// Mitsubishi GX Works2 project: BookEX6_35 Struct   PLC: Q13UDV

// global labels: Global
VAR_GLOBAL
  bVar0 AT M5000 : BOOL;
  abArray0 AT M5010 : ARRAY [0..49] OF BOOL;
  sStr0 AT D5000 : STRING[199];
  sStr1 AT D5100 : STRING[199];
  sStr2 AT D5200 : STRING[199];
  sStr3 AT D5300 : STRING[199];
  sStr4 AT D5400 : STRING[199];
  sStr5 AT D5500 : STRING[199];
  sStr6 AT D5600 : STRING[199];
  sStr7 AT D5700 : STRING[199];
  sStr8 AT D5800 : STRING[199];
  sStr9 AT D5900 : STRING[199];
  iVar0 AT D4500 : INT;
  iVar1 AT D4501 : INT;
  iVar2 AT D4502 : INT;
  iVar3 AT D4503 : INT;
  iVar4 AT D4504 : INT;
  iVar5 AT D4505 : INT;
  iVar6 AT D4506 : INT;
  iVar7 AT D4507 : INT;
  iVar8 AT D4508 : INT;
  iVar9 AT D4509 : INT;
  dVar0 AT D4510 : DINT;
  dVar1 AT D4512 : DINT;
  dVar2 AT D4514 : DINT;
  dVar3 AT D4516 : DINT;
  dVar4 AT D4518 : DINT;
  dVar5 AT D4520 : DINT;
  dVar6 AT D4522 : DINT;
  dVar7 AT D4524 : DINT;
  dVar8 AT D4526 : DINT;
  dVar9 AT D4528 : DINT;
  wVar0 AT D4530 : WORD;
  wVar1 AT D4531 : WORD;
  wVar2 AT D4532 : WORD;
  wVar3 AT D4533 : WORD;
  wVar4 AT D4534 : WORD;
  wVar5 AT D4535 : WORD;
  wVar6 AT D4536 : WORD;
  wVar7 AT D4537 : WORD;
  wVar8 AT D4538 : WORD;
  wVar9 AT D4539 : WORD;
  dwVar0 AT D4540 : DWORD;
  dwVar1 AT D4542 : DWORD;
  dwVar2 AT D4544 : DWORD;
  dwVar3 AT D4546 : DWORD;
  dwVar4 AT D4548 : DWORD;
  dwVar5 AT D4550 : DWORD;
  dwVar6 AT D4552 : DWORD;
  dwVar7 AT D4554 : DWORD;
  dwVar8 AT D4556 : DWORD;
  dwVar9 AT D4558 : DWORD;
  fsVar0 AT D4560 : REAL;
  fsVar1 AT D4562 : REAL;
  fsVar2 AT D4564 : REAL;
  fsVar3 AT D4566 : REAL;
  fsVar4 AT D4568 : REAL;
  fsVar5 AT D4570 : REAL;
  fsVar6 AT D4572 : REAL;
  fsVar7 AT D4574 : REAL;
  fsVar8 AT D4576 : REAL;
  fsVar9 AT D4578 : REAL;
  fdVar0 AT D4580 : LREAL;
  tTime0 AT D4620 : TIME;
  tTime1 AT D4622 : TIME;
  tTime2 AT D4624 : TIME;
  tTime3 AT D4626 : TIME;
  tTime4 AT D4628 : TIME;
  tTime5 AT D4630 : TIME;
  tTime6 AT D4632 : TIME;
  tTime7 AT D4634 : TIME;
  tTime8 AT D4636 : TIME;
  tTime9 AT D4638 : TIME;
  tTime10 AT D4640 : TIME;
  bVar1 AT M5001 : BOOL;
  bVar2 AT M5002 : BOOL;
  bVar3 AT M5003 : BOOL;
  bVar4 AT M5004 : BOOL;
  bVar5 AT M5005 : BOOL;
  bVar6 AT M5006 : BOOL;
  bVar7 AT M5007 : BOOL;
  bVar8 AT M5008 : BOOL;
  bVar9 AT M5009 : BOOL;
  abArray1 AT M5060 : ARRAY [0..49] OF BOOL;
  abArray2 AT M5110 : ARRAY [0..49] OF BOOL;
  abArray3 AT M5160 : ARRAY [0..49] OF BOOL;
  abArray4 AT M5210 : ARRAY [0..49] OF BOOL;
  abArray5 AT M5260 : ARRAY [0..49] OF BOOL;
  abArray6 AT M5310 : ARRAY [0..49] OF BOOL;
  abArray7 AT M5360 : ARRAY [0..49] OF BOOL;
  abArray8 AT M5410 : ARRAY [0..49] OF BOOL;
  abArray9 AT M5460 : ARRAY [0..49] OF BOOL;
  fdVar1 AT D4584 : LREAL;
  fdVar2 AT D4588 : LREAL;
  fdVar3 AT D4592 : LREAL;
  fdVar4 AT D4596 : LREAL;
  fdVar5 AT D4600 : LREAL;
  fdVar6 AT D4604 : LREAL;
  fdVar7 AT D4608 : LREAL;
  fdVar8 AT D4612 : LREAL;
  fdVar9 AT D4616 : LREAL;
  afsPen0 AT D2000 : ARRAY [0..499] OF REAL;
  afsPen1 AT D3000 : ARRAY [0..499] OF REAL;
END_VAR
// user libraries (not included): HMI

PROGRAM ExBREAK
(* structured ladder/FBD written out as ST: instructions are called as NAME(EN, inputs, outputs); _pN, _eN, _tN stand for wires *)
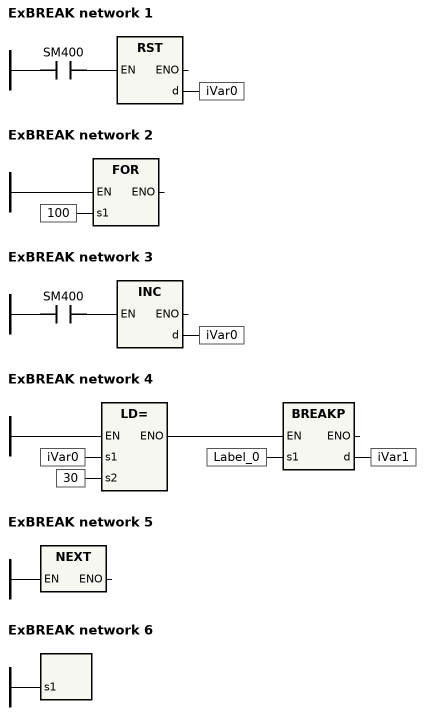
(* network 1 *)
RST(SM400, iVar0);
(* network 2 *)
FOR(TRUE, 100);
(* network 3 *)
INC(SM400, iVar0);
(* network 4 *)
_e1 := LD=(TRUE, iVar0, 30);
BREAKP(_e1, Label_0, iVar1);
(* network 5 *)
NEXT(TRUE);
(* network 6 Label_0: *)
(* element kind 10  <- TRUE *)
END_PROGRAM

PROGRAM ExCALL
(* structured ladder/FBD written out as ST: instructions are called as NAME(EN, inputs, outputs); _pN, _eN, _tN stand for wires *)
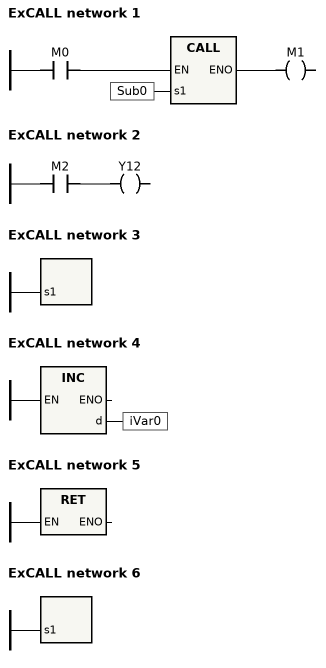
(* network 1 *)
_e1 := CALL(M0, Sub0);
M1 := _e1;
(* network 2 *)
Y12 := M2;
(* network 3 *)
(* element kind 10  <- TRUE *)
(* network 4 Sub0: *)
INC(TRUE, iVar0);
(* network 5 *)
RET(TRUE);
(* network 6 *)
(* element kind 10  <- TRUE *)
END_PROGRAM

PROGRAM ExCALL2
(* structured ladder/FBD written out as ST: instructions are called as NAME(EN, inputs, outputs); _pN, _eN, _tN stand for wires *)
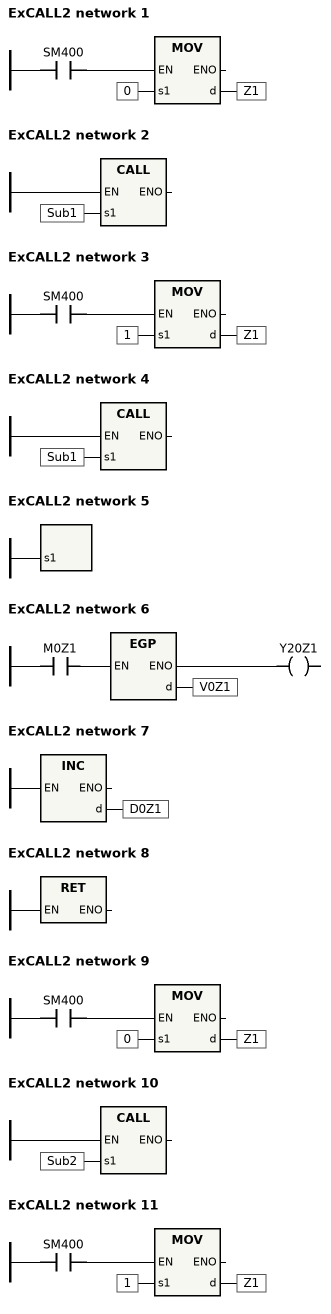
(* network 1 *)
MOV(SM400, 0, Z1);
(* network 2 *)
CALL(TRUE, Sub1);
(* network 3 *)
MOV(SM400, 1, Z1);
(* network 4 *)
CALL(TRUE, Sub1);
(* network 5 *)
(* element kind 10  <- TRUE *)
(* network 6 Sub1: *)
_e1 := EGP(M0Z1, V0Z1);
Y20Z1 := _e1;
(* network 7 *)
INC(TRUE, D0Z1);
(* network 8 *)
RET(TRUE);
(* network 9 *)
MOV(SM400, 0, Z1);
(* network 10 *)
CALL(TRUE, Sub2);
(* network 11 *)
MOV(SM400, 1, Z1);
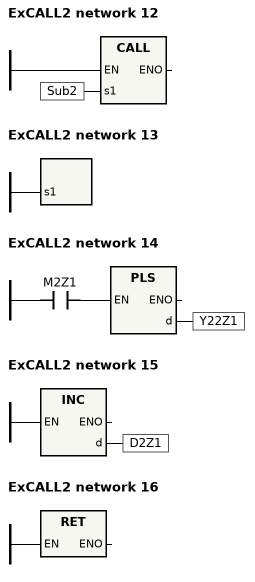
(* network 12 *)
CALL(TRUE, Sub2);
(* network 13 *)
(* element kind 10  <- TRUE *)
(* network 14 Sub2: *)
PLS(M2Z1, Y22Z1);
(* network 15 *)
INC(TRUE, D2Z1);
(* network 16 *)
RET(TRUE);
END_PROGRAM

PROGRAM ExCALL3
VAR
  Mov4INT_1 : Mov4INT;
END_VAR
(* structured ladder/FBD written out as ST: instructions are called as NAME(EN, inputs, outputs); _pN, _eN, _tN stand for wires *)
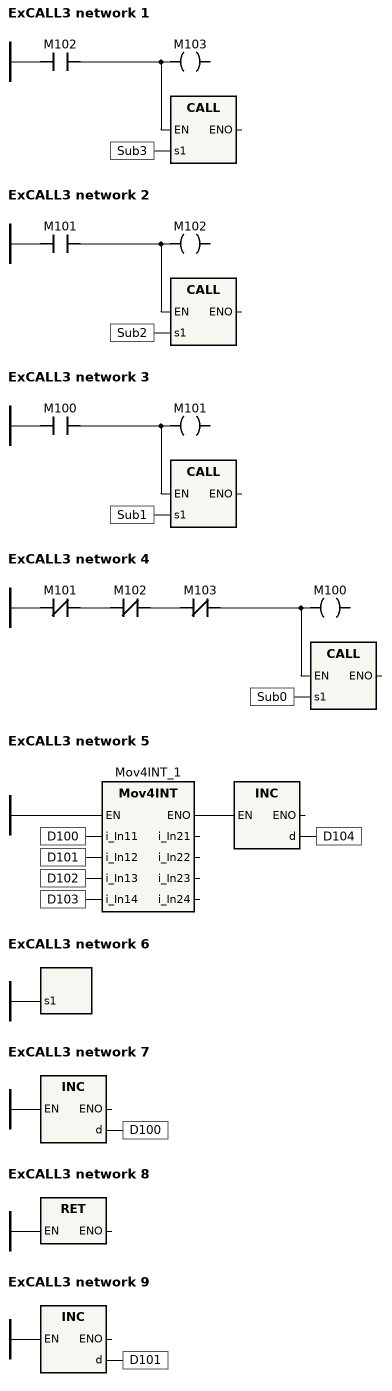
(* network 1 *)
M103 := M102;
CALL(M102, Sub3);
(* network 2 *)
M102 := M101;
CALL(M101, Sub2);
(* network 3 *)
M101 := M100;
CALL(M100, Sub1);
(* network 4 *)
_p1 := NOT M101 AND NOT M102 AND NOT M103;
M100 := _p1;
CALL(_p1, Sub0);
(* network 5 *)
Mov4INT_1(EN := TRUE, i_In11 := D100, i_In12 := D101, i_In13 := D102, i_In14 := D103);
INC(Mov4INT_1.ENO, D104);
(* network 6 *)
(* element kind 10  <- TRUE *)
(* network 7 Sub0: *)
INC(TRUE, D100);
(* network 8 *)
RET(TRUE);
(* network 9 Sub1: *)
INC(TRUE, D101);
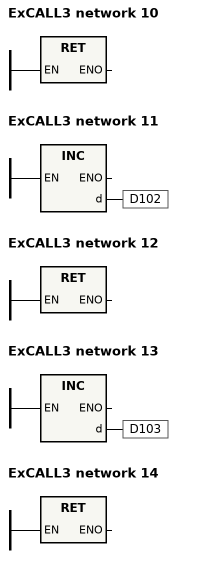
(* network 10 *)
RET(TRUE);
(* network 11 Sub2: *)
INC(TRUE, D102);
(* network 12 *)
RET(TRUE);
(* network 13 Sub3: *)
INC(TRUE, D103);
(* network 14 *)
RET(TRUE);
END_PROGRAM

PROGRAM ExCOM
END_PROGRAM

PROGRAM ExFOR
(* structured ladder/FBD written out as ST: instructions are called as NAME(EN, inputs, outputs); _pN, _eN, _tN stand for wires *)
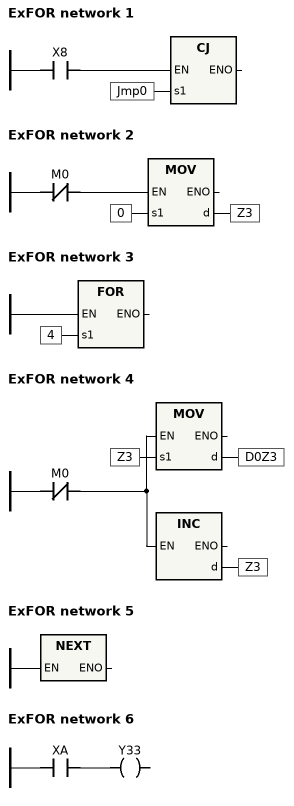
(* network 1 *)
CJ(X8, Jmp0);
(* network 2 *)
MOV(NOT M0, 0, Z3);
(* network 3 *)
FOR(TRUE, 4);
(* network 4 *)
_p1 := NOT M0;
MOV(_p1, Z3, D0Z3);
INC(_p1, Z3);
(* network 5 *)
NEXT(TRUE);
(* network 6 Jmp0: *)
Y33 := XA;
END_PROGRAM

PROGRAM ExFOR2
(* structured ladder/FBD written out as ST: instructions are called as NAME(EN, inputs, outputs); _pN, _eN, _tN stand for wires *)
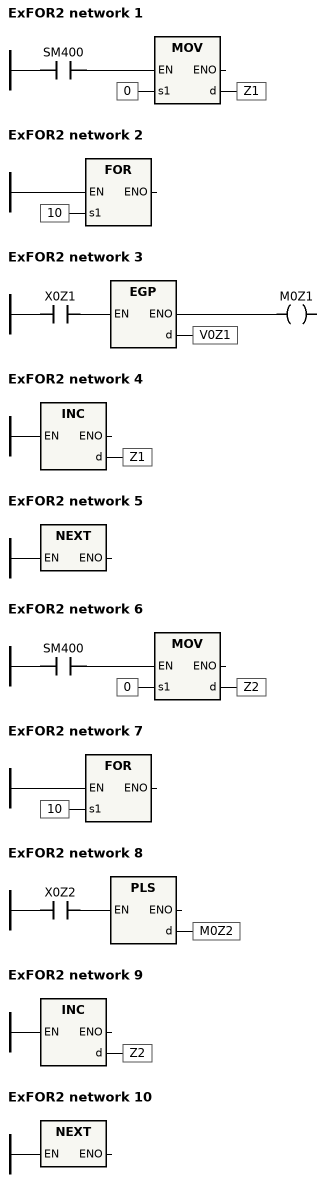
(* network 1 *)
MOV(SM400, 0, Z1);
(* network 2 *)
FOR(TRUE, 10);
(* network 3 *)
_e1 := EGP(X0Z1, V0Z1);
M0Z1 := _e1;
(* network 4 *)
INC(TRUE, Z1);
(* network 5 *)
NEXT(TRUE);
(* network 6 *)
MOV(SM400, 0, Z2);
(* network 7 *)
FOR(TRUE, 10);
(* network 8 *)
PLS(X0Z2, M0Z2);
(* network 9 *)
INC(TRUE, Z2);
(* network 10 *)
NEXT(TRUE);
END_PROGRAM
